// TwinCAT 3 PLC project OwiePLC1
// ProgramVersion: 3.1.4024.0
// libraries:
//   Tc2_Standard, * (Beckhoff Automation GmbH)
//   Tc2_System, * (Beckhoff Automation GmbH)
//   Tc3_Module, * (Beckhoff Automation GmbH)
// project tree:
//   DUTs/ AxisStatus.TcDUT, Motor.TcDUT, MotorProxy.TcDUT, ST_ComboboxEntry.TcDUT
//   GVLs/ GVL.TcGVL
//   / PlcTask.TcTTO
//   POUs/ MAIN.TcPOU, TransferMotorDataToProxy.TcPOU

CONFIGURATION OwiePLC1
    RESOURCE PLC ON TwinCAT3
        TASK PlcTask(INTERVAL := T#10ms, PRIORITY := 20);
        PROGRAM MAIN WITH PlcTask : MAIN;
    END_RESOURCE
END_CONFIGURATION

// ---- DUTs/AxisStatus.TcDUT
{attribute 'qualified_only'}
{attribute 'strict'}
TYPE AxisStatus :
(
	Ready,
	STO_Active,
	Faulted
);
END_TYPE

// ---- DUTs/Motor.TcDUT
TYPE Motor :
STRUCT	
	name: STRING;
	motorId: INT;
	isAxisSelected: BOOL;
	
	encoder: REAL;
	status: AxisStatus;
END_STRUCT
END_TYPE

// ---- DUTs/MotorProxy.TcDUT
TYPE MotorProxy :
STRUCT
	motorPtr: POINTER TO Motor;
	IsAxisSelected: BOOL;
	flagOne: BOOL;
	encoder: REAL;
	status: AxisStatus;
END_STRUCT


END_TYPE

// ---- DUTs/ST_ComboboxEntry.TcDUT
TYPE ST_ComboboxEntry:
STRUCT
    id : INT;
    text : WSTRING;
    value : INT;
END_STRUCT
END_TYPE

// ---- GVLs/GVL.TcGVL
{attribute 'qualified_only'}
VAR_GLOBAL
	
	px: MotorProxy;
	motors: ARRAY[0..3] OF Motor;
END_VAR

// ---- POUs/MAIN.TcPOU
PROGRAM MAIN
VAR
	selectedIndex: INT := 0;
	px: MotorProxy;
	motors: ARRAY[0..3] OF Motor;
	
	
	aComboboxEntries : ARRAY [0..5] OF ST_ComboboxEntry;

	
	
	
END_VAR


	aComboboxEntries[0].id:=0;
	aComboboxEntries[0].text:="Motor One";
	aComboboxEntries[0].value:=0;
	
	
	






//	GVL.motors[0].name := "One";
	motors[0].motorId := 1;
	motors[0].isAxisSelected := 1;
	motors[0].encoder := 0.012;
	motors[0].status := AxisStatus.Ready;
	
	//GVL.motors[1].name := "Two";
	motors[1].motorId := 2;
	motors[1].isAxisSelected := 1;
	motors[1].encoder := 0.012;
	motors[1].status := AxisStatus.Ready;
	
	//GVL.motors[2].name := "Three";
	motors[2].motorId := 3;
	motors[2].isAxisSelected := 1;
	motors[2].encoder := 0.012;
	motors[2].status := AxisStatus.Ready;

END_PROGRAM

// ---- POUs/TransferMotorDataToProxy.TcPOU
FUNCTION TransferMotorDataToProxy : BOOL
VAR_INPUT
	mp: POINTER TO MotorProxy;
	
END_VAR
VAR
	
	prox: MotorProxy;
	moto: Motor;



END_VAR


	
	prox := mp^;
	mp := prox.motorPtr^;
	
	prox.encoder := moto.encoder;
	prox.IsAxisSelected := moto.isAxisSelected;
	prox.status := moto.status;

END_FUNCTION
